Staubli VAL3: getSize.pgx

public program getSize(num& x_nSize[])
begin
  // size
  x_nSize=size(saveInOut:dInput)
end
